INTERFACE ITF_Mover

METHOD GetMaxVelo : LREAL
VAR_INPUT
END_VAR
END_METHOD

METHOD SetMaxVelo : BOOL
VAR_INPUT
	MaxVelocity : LREAL;
END_VAR
END_METHOD

END_INTERFACE

(* stored: Version 1.1.0.1, ProductVersion 3.1.4024.12
   Itf ITF_Mover: Id {32d35547-7ce1-48b8-89d6-1e503b2efd40}
   Method GetMaxVelo: Id {7d7f9943-ad14-49e5-b77f-4592447f9233}
   Method SetMaxVelo: Id {4d4c8ec2-564a-4e49-9412-d89887fcf940} *)
